FUNCTION_BLOCK FB_RoughPump
VAR_INPUT
END_VAR
VAR_OUTPUT
END_VAR
VAR_IN_OUT
	stVolInlet	:	ST_Volume;
	stPump	:	ST_MechPump;
END_VAR
VAR
END_VAR

(* 
Roughing pump

A roughing pump removes matter from the inlet at a specified
rate.

A. Wallace, 2016-2-28
*)

IF stPump.i_xRun THEN//Press the Pump Run button
	// drop the pressure by a small percentage of the total pressure
	stVolInlet.rPressure := MAX( stVolInlet.rPressure*(1-stPump.rMRE/stVolInlet.rVolume), stPump.rBasePress);
END_IF

END_FUNCTION_BLOCK

(* stored: Version 1.1.0.1, ProductVersion 3.1.4020.12
   POU FB_RoughPump: Id {1c0a7f67-206d-4f00-a16d-b41dffef9f3c}, SpecialFunc None *)
